# EPICS autosave request: elmitecLEEM/leem-PSValue_settings.req
$(P)$(Q):TGL:FREQ
$(P)$(Q):TGL:HI
$(P)$(Q):TGL:LO
$(P)$(Q):TWV
$(P)$(Q):TWVH
$(P)$(Q):TWVL
$(P)$(Q):TWVM
